PROGRAM PRG_IM1L0_XTES
VAR
    {attribute 'pytmc' := '
        pv: IM1L0:XTES
        io: io
    '}
    {attribute 'TcLinkTo' := '.bZoomEndFwd := TIIB[IM1L0-EL1088]^Channel 1^Input;
                              .bZoomEndBwd := TIIB[IM1L0-EL1088]^Channel 2^Input;
                              .bFocusEndFwd := TIIB[IM1L0-EL1088]^Channel 3^Input;
                              .bFocusEndBwd := TIIB[IM1L0-EL1088]^Channel 4^Input;
                              .fbOpal.bOpalPower := TIIB[IM1L0-EL2004]^Channel 2^Output;
                              .fbLED.bLedPower := TIIB[IM1L0-EL2004]^Channel 3^Output'}
    fbIM1L0: FB_XPIM;
    {attribute 'pytmc' := '
        pv: IM1L0:XTES:FLOW_OK
        field: ZNAM LOW
        field: ONAM OK
    '}
    {attribute 'TcLinkTo' := 'TIIB[IM1L0-EL7342]^DCM Status Channel 1^Status^Digital input 1'}
    bIM1L0FlowOk AT %I*: BOOL;
    {attribute 'TcLinkTo' := '.Status := TIIB[IM1L0-EL6002]^COM TxPDO-Map Inputs Channel 1^Status;
                              .D[0] := TIIB[IM1L0-EL6002]^COM TxPDO-Map Inputs Channel 1^Data In 0;
                              .D[1] := TIIB[IM1L0-EL6002]^COM TxPDO-Map Inputs Channel 1^Data In 1;
                              .D[2] := TIIB[IM1L0-EL6002]^COM TxPDO-Map Inputs Channel 1^Data In 2;
                              .D[3] := TIIB[IM1L0-EL6002]^COM TxPDO-Map Inputs Channel 1^Data In 3;
                              .D[4] := TIIB[IM1L0-EL6002]^COM TxPDO-Map Inputs Channel 1^Data In 4;
                              .D[5] := TIIB[IM1L0-EL6002]^COM TxPDO-Map Inputs Channel 1^Data In 5;
                              .D[6] := TIIB[IM1L0-EL6002]^COM TxPDO-Map Inputs Channel 1^Data In 6;
                              .D[7] := TIIB[IM1L0-EL6002]^COM TxPDO-Map Inputs Channel 1^Data In 7;
                              .D[8] := TIIB[IM1L0-EL6002]^COM TxPDO-Map Inputs Channel 1^Data In 8;
                              .D[9] := TIIB[IM1L0-EL6002]^COM TxPDO-Map Inputs Channel 1^Data In 9;
                              .D[10] := TIIB[IM1L0-EL6002]^COM TxPDO-Map Inputs Channel 1^Data In 10;
                              .D[11] := TIIB[IM1L0-EL6002]^COM TxPDO-Map Inputs Channel 1^Data In 11;
                              .D[12] := TIIB[IM1L0-EL6002]^COM TxPDO-Map Inputs Channel 1^Data In 12;
                              .D[13] := TIIB[IM1L0-EL6002]^COM TxPDO-Map Inputs Channel 1^Data In 13;
                              .D[14] := TIIB[IM1L0-EL6002]^COM TxPDO-Map Inputs Channel 1^Data In 14;
                              .D[15] := TIIB[IM1L0-EL6002]^COM TxPDO-Map Inputs Channel 1^Data In 15;
                              .D[16] := TIIB[IM1L0-EL6002]^COM TxPDO-Map Inputs Channel 1^Data In 16;
                              .D[17] := TIIB[IM1L0-EL6002]^COM TxPDO-Map Inputs Channel 1^Data In 17;
                              .D[18] := TIIB[IM1L0-EL6002]^COM TxPDO-Map Inputs Channel 1^Data In 18;
                              .D[19] := TIIB[IM1L0-EL6002]^COM TxPDO-Map Inputs Channel 1^Data In 19;
                              .D[20] := TIIB[IM1L0-EL6002]^COM TxPDO-Map Inputs Channel 1^Data In 20;
                              .D[21] := TIIB[IM1L0-EL6002]^COM TxPDO-Map Inputs Channel 1^Data In 21'}
    stEL6In AT %I*: EL6InData22b;
    {attribute 'TcLinkTo' := '.Ctrl := TIIB[IM1L0-EL6002]^COM RxPDO-Map Outputs Channel 1^Ctrl;
                              .D[0] := TIIB[IM1L0-EL6002]^COM RxPDO-Map Outputs Channel 1^Data Out 0;
                              .D[1] := TIIB[IM1L0-EL6002]^COM RxPDO-Map Outputs Channel 1^Data Out 1;
                              .D[2] := TIIB[IM1L0-EL6002]^COM RxPDO-Map Outputs Channel 1^Data Out 2;
                              .D[3] := TIIB[IM1L0-EL6002]^COM RxPDO-Map Outputs Channel 1^Data Out 3;
                              .D[4] := TIIB[IM1L0-EL6002]^COM RxPDO-Map Outputs Channel 1^Data Out 4;
                              .D[5] := TIIB[IM1L0-EL6002]^COM RxPDO-Map Outputs Channel 1^Data Out 5;
                              .D[6] := TIIB[IM1L0-EL6002]^COM RxPDO-Map Outputs Channel 1^Data Out 6;
                              .D[7] := TIIB[IM1L0-EL6002]^COM RxPDO-Map Outputs Channel 1^Data Out 7;
                              .D[8] := TIIB[IM1L0-EL6002]^COM RxPDO-Map Outputs Channel 1^Data Out 8;
                              .D[9] := TIIB[IM1L0-EL6002]^COM RxPDO-Map Outputs Channel 1^Data Out 9;
                              .D[10] := TIIB[IM1L0-EL6002]^COM RxPDO-Map Outputs Channel 1^Data Out 10;
                              .D[11] := TIIB[IM1L0-EL6002]^COM RxPDO-Map Outputs Channel 1^Data Out 11;
                              .D[12] := TIIB[IM1L0-EL6002]^COM RxPDO-Map Outputs Channel 1^Data Out 12;
                              .D[13] := TIIB[IM1L0-EL6002]^COM RxPDO-Map Outputs Channel 1^Data Out 13;
                              .D[14] := TIIB[IM1L0-EL6002]^COM RxPDO-Map Outputs Channel 1^Data Out 14;
                              .D[15] := TIIB[IM1L0-EL6002]^COM RxPDO-Map Outputs Channel 1^Data Out 15;
                              .D[16] := TIIB[IM1L0-EL6002]^COM RxPDO-Map Outputs Channel 1^Data Out 16;
                              .D[17] := TIIB[IM1L0-EL6002]^COM RxPDO-Map Outputs Channel 1^Data Out 17;
                              .D[18] := TIIB[IM1L0-EL6002]^COM RxPDO-Map Outputs Channel 1^Data Out 18;
                              .D[19] := TIIB[IM1L0-EL6002]^COM RxPDO-Map Outputs Channel 1^Data Out 19;
                              .D[20] := TIIB[IM1L0-EL6002]^COM RxPDO-Map Outputs Channel 1^Data Out 20;
                              .D[21] := TIIB[IM1L0-EL6002]^COM RxPDO-Map Outputs Channel 1^Data Out 21'}
    stEL6Out AT %Q*: EL6OutData22b;

    fbStateSetup: FB_StateSetupHelper;
    stDefault: ST_PositionState := (
        fVelocity := 1,
        bMoveOk := TRUE,
        bValid := TRUE
    );
END_VAR


fbStateSetup(stPositionState:=stDefault, bSetDefault:=TRUE);
fbStateSetup(stPositionState:=fbIM1L0.stOut, fPosition:=0,          sPmpsState:='IM1L0:XTES-OUT');
fbStateSetup(stPositionState:=fbIM1L0.stYag, fPosition:=-86.65,     sPmpsState:='IM1L0:XTES-YAG');
fbStateSetup(stPositionState:=fbIM1L0.stDiamond, fPosition:=-56.65, sPmpsState:='IM1L0:XTES-DIAMOND');
fbStateSetup(stPositionState:=fbIM1L0.stReticle, fPosition:=-26.65, sPmpsState:='IM1L0:XTES-RETICLE');

fbIM1L0(
    fbArbiter := GVL.fbArbiter,
    fbFFHWO := GVL.fbFastFaultOutput1a,
    stYStage := Main.M20,
    stZoomStage := Main.M21,
    stFocusStage := Main.M22,
    stEl6In := stEL6In,
    stEl6Out := stEl6Out,
    sDeviceName := 'IM1L0:XTES',
    sTransitionKey := 'IM1L0:XTES-TRANSITION',
    bEnableMotion := TRUE,
    bEnableBeamParams := TRUE,
    bEnablePositionLimits := TRUE,
);

END_PROGRAM

(* stored: Version 1.1.0.1
   POU PRG_IM1L0_XTES: Id {dc3548d0-1688-4ec2-b4ae-fd34a5036e7d}, SpecialFunc None *)
